FUNCTION_BLOCK T_MobjectQueue_AddItem_AddsItem EXTENDS T_UnitTestBase
VAR_INPUT
END_VAR
VAR_OUTPUT
END_VAR
VAR
	Queue : Queue;
	queueLength : DINT;
	item : INT := 1;
END_VAR

Queue.AddItem(item);
queueLength := Queue.Count;
TestFinished();

END_FUNCTION_BLOCK

(* stored: Version 1.1.0.1, ProductVersion 3.1.4024.12
   POU T_MobjectQueue_AddItem_AddsItem: Id {5d9a6006-e93c-407c-bc1a-e901a602b81a}, SpecialFunc None *)
